Staubli VAL3: start.pgx

public program start()
begin

  // The start function's purpose is to make sure everything is reset and setup
  // It starts by initing a few variables the program uses then moving the arm to the homePoint


  //initing a few variables
  nBuffer=0
  nNum=0
  nFailCounter=0
  bDetectInput=false
  sInput=""

  //Set the arm at the homePoint
  movej(homePoint,tClaw,nom_speed)
  waitEndMove()
  //call enablePowerTest()
  call detectInput()
end
